# EPICS substitutions: mc02/db/fb_epid.substitutions
file "db/fb_epid.db" {
	    pattern { Sys , Dev , IN , OUT , MODE , CALC ,
		          PERMIT1 , PERMIT2 , PERMIT3, PERMIT4 ,
				  PREC , EGU , IEGU , OEGU }
		{ "XF:23ID2-OP", "{FBck}", "XF:23ID2-BI{ExitSlt-Cam:1}Stats1:CX_RBV CPP",
		  "XF:23IDA-OP:2{Mir:1A-Ax:FPit}Mtr_POS_SP PP" , "PID" , "A&B" ,
		  "" , "" , "" , "" ,
		  "3" , "" , "pix" , "urad" }
}
